// TIA Portal V16 export
// export: Created 2023-05-08T20:48:17.490425Z, ExportSetting WithDefaults, DisplayName Totally Integrated Automation Portal, DisplayVersion V16 Update 6, DisplayName TIA Portal Version Control Interface, DisplayVersion V16 Update 2, DisplayName TIA Portal Openness, DisplayVersion V16 Update 6, DisplayName STEP 7 Professional, DisplayVersion V16 Update 6, DisplayName STEP 7 Safety, DisplayVersion V16, DisplayName WinCC Advanced, DisplayVersion V16 Update 6
FUNCTION "MHJ-PLC-Lab-Function-S71500-NextInputArea" : Void   // FC2, SCL
{ S7_Optimized_Access := 'TRUE' }
VERSION : 0.1
// stored: AutoNumber true, IsIECCheckEnabled false, SetENOAutomatically false, UDAEnableTagReadback false
   VAR_INPUT
      MinDiByte : Int;
      MaxDiByte : Int;
   END_VAR
   VAR_TEMP
      Value : Byte;
      ForCounter : Int;
      MaxDiByteTemp : Int;
      MinDiByteTemp : Int;
   END_VAR
BEGIN


   #MaxDiByteTemp := -1;
   IF #MaxDiByte < 463 THEN
       #MaxDiByteTemp := #MaxDiByte;
   END_IF;

   #MinDiByteTemp := -1;
   IF #MaxDiByteTemp >= #MinDiByte & #MinDiByte >= 0 THEN
       #MinDiByteTemp := #MinDiByte;
   END_IF;

   IF #MaxDiByteTemp >= 0 & #MinDiByte >= 0 THEN
       FOR #ForCounter := #MinDiByteTemp TO #MaxDiByteTemp DO
           #Value := PEEK(area := 16#1,
                          dbNumber := 0,
                          byteOffset := #ForCounter);
           POKE(area := 16#81,
                dbNumber := 0,
                byteOffset := #ForCounter,
                value := #Value);
       END_FOR;

   END_IF;
END_FUNCTION
